KUKA KRL program: FlexPumpOff.src

&ACCESS RVO3
&PARAM EDITMASK = *
&PARAM TEMPLATE = C:\KRC\Roboter\Template\vorgabe
DEF FlexPumpOff( )

;************************************************
;              CNC Robotics Ltd
;              www.cncrobotics.co.uk
;************************************************
;     Contact: helpdesk@cncrobotics.co.uk
;     Date: 25/09/23
;     Version: 0.8.38
;     Date: 25/09/23
;     Version: 0.9.46
;************************************************
; Description: Routine to turn off the Flex Pump
; 			   Off
;************************************************

WAIT SEC 0
oTrackLubrication = FALSE

END
